Universal Robots PolyScope program: AlvarezZavaleta-LuisAlberto-P5.urp

Program AlvarezZavaleta-LuisAlberto-P5 (installation=default directory=/programs/usbdisk_0 createdIn=5.14.5 lastSavedIn=5.14.5 robotSerialNumber=20225300689)
Calibrated DH parameters: a=[-0.000069, -0.212707, -0.211705, 0.000184, -0.000164, 0]; d=[0.151915, 16.812457, -12.99464, -3.686678, 0.08547, 0.092229]; alpha=[1.56993, 0.007145, 0.006979, 1.572433, -1.572917, 0]; deltaTheta=[0, 0.514054, 5.89431, -0.125193, 0.000032, 0]
InitVariablesNode
BeforeStart
  Set DigitalOutput pin=digital_out[0]; digitalValue=1
  Script: freedrive_mode(freeAxes=[1,1,1,0,0,0])
  Popup Message (haltProgram=false message=Define First Point P1 inputType=Text)
  P1 := get_actual_tcp_pose()
  Popup Message (haltProgram=false message=Define Second Point P2 inputType=Text)
  P2 := get_actual_tcp_pose()
  Popup Message (haltProgram=false message=Define Pini inputType=Text)
  Pini := get_actual_tcp_pose()
  Script: end_freedrive_mode()
  n :=  (valueSource=Operator message=Numero de impactos por linea valueType=Integer)
  l :=  (valueSource=Operator message=Longitud a ensayar(mm) valueType=Integer)
  Nrep :=  (valueSource=Operator message=Num Repeticiones linea valueType=Integer)
  d_lat :=  (valueSource=Operator message=Distancia ensayo lateral(mm) valueType=Integer)
  Nrep_lat :=  (valueSource=Operator message=Num Repeticiones linea lateral valueType=Integer)
Robot Program (runOnlyOnce=true)
  distPunto := l/(n*1000)
  direction := [P2[0]-P1[0],P2[1]-P1[0]]
  direction := [direction[0]/(norm(direction)),direction[1]/(norm(direction))]
  SuppressedNode
    direction := [0,1]
  distance := p[0,0,45/1000,0,0,0]
  Pini := pose_add(Pini, distance)
  Pbase := Pini
  i := 0
  Loop While (checkContinuously=false) expression=i<Nrep
    j := 0
    Loop While (checkContinuously=false) expression=j<n+1
      distance := p[distPunto*j*direction[0],distPunto*j*direction[1],0,0,0,0]
      Ppoint := pose_add(Pbase, distance)
      MoveJ speed 60 deg/s, acceleration 80 deg/s^2 (useActiveTCP=true) feature=Base
        Waypoint Variable (Variable): variable=Ppoint
      Call TestPoint
      j := j+1
    i := i+1
  i := 0
  'Vector perpendicular dist*z siendo z (0,0,1,0,0,0)'
  distance := p[direction[1]*d_lat/1000,-direction[0]*d_lat/1000,0,0,0,0]
  Pbase := pose_add(Pini, distance)
  Loop While (checkContinuously=false) expression=i<Nrep_lat
    j := 0
    Loop While (checkContinuously=false) expression=j<n+1
      distance := p[distPunto*j*direction[0],distPunto*j*direction[1],0,0,0,0]
      Ppoint := pose_add(Pbase, distance)
      MoveJ speed 60 deg/s, acceleration 80 deg/s^2 (useActiveTCP=true) feature=Base
        Waypoint Variable (Variable): variable=Ppoint
      Call TestPoint
      j := j+1
    i := i+1
  i := 0
  'Vector perpendicular contrario dist*z siendo z (0,0,1,0,0,0)'
  distance := p[-direction[1]*d_lat/1000,direction[0]*d_lat/1000,0,0,0,0]
  Pbase := pose_add(Pini, distance)
  Loop While (checkContinuously=false) expression=i<Nrep_lat
    j := 0
    Loop While (checkContinuously=false) expression=j<n+1
      distance := p[distPunto*j*direction[0],distPunto*j*direction[1],0,0,0,0]
      Ppoint := pose_add(Pbase, distance)
      MoveJ speed 60 deg/s, acceleration 80 deg/s^2 (useActiveTCP=true) feature=Base
        Waypoint Variable (Variable): variable=Ppoint
      Call TestPoint
      j := j+1
    i := i+1
  MoveJ speed 60 deg/s, acceleration 80 deg/s^2 (useActiveTCP=true) feature=Base
    Waypoint Variable (Variable): variable=Pini
SubProgram -> TestPoint
SubProgram TestPoint (keepSynchronizedWithDisk=false)
  Set DigitalOutput pin=digital_out[2]; digitalValue=0
  Wait Sleep waitTime=0.1
  Set DigitalOutput pin=digital_out[0]; digitalValue=0
  Set DigitalOutput pin=digital_out[4]; digitalValue=1
  Wait Sleep waitTime=0.4
  Set DigitalOutput pin=digital_out[4]; digitalValue=0
  Wait Sleep waitTime=0.1
